{attribute 'linkalways'} 
{attribute 'no_explicit_call' := 'This FB is a CLASS and must be accessed using methods or properties'}
{attribute 'enable_dynamic_creation'}
FUNCTION_BLOCK Node_F_VN_ContourMoments EXTENDS VisionNode
VAR
    ipContour : _ITcVnContainer;
    stMoments : _TcVnMoments;
    hrPrev : _HRESULT(S_OK);
	hresult : _HRESULT(S_OK);
END_VAR

METHOD PUBLIC  Clone : I_Node
VAR
	pNode : POINTER TO Node_F_VN_ContourMoments;
END_VAR
pNode := __NEW(Node_F_VN_ContourMoments);
Clone := pNode^;
END_METHOD

METHOD FB_init : BOOL
VAR_INPUT
	bInitRetains : BOOL; // if TRUE, the retain variables are initialized (warm start / cold start)
	bInCopyCode : BOOL;  // if TRUE, the instance afterwards gets moved into the copy code (online change)
END_VAR
AddInput('ipContour', ipContour);
AddInput('hrPrev', hrPrev);
AddOutput('stMoments', stMoments);
AddOutput('hresult',hresult);
END_METHOD

METHOD PROTECTED OnExecute
hresult.Value := F_VN_ContourMoments(
	ipContour := ipContour.Value,
    stMoments := stMoments.Value,
	hrPrev:= hrPrev.Value);
END_METHOD

METHOD PUBLIC PreExecutionCheck
VAR_INPUT
	Check : I_PreExecutionChecks;
END_VAR
Check.IsTrue(ipContour.IsValid, 'ipContour must be a valid container');
Check.IsTrue((ipContour.IsType(TC_GLOBAL_CONST_LIST.ContainerType_Vector_TcVnPoint2_DINT) OR
              ipContour.IsType(TC_GLOBAL_CONST_LIST.ContainerType_Vector_TcVnPoint2_REAL)),
              'ipContour contains incorrect type');
END_METHOD

END_FUNCTION_BLOCK

(* stored: Version 1.1.0.1, ProductVersion 3.1.4026.13
   POU Node_F_VN_ContourMoments: Id {f1f8bd5b-fb7d-09f7-3cd6-ff0fb48e97c2}, SpecialFunc None
   Folder Constructor: Id {1bb0c863-8b3a-0ade-09be-99531624ab88}
   Method Clone: Id {44b8e371-313f-0c62-0852-1be687f9b1b8}
   Method FB_init: Id {a5f4f229-2a67-036c-16f2-5f92c8fbdc9f}
   Method OnExecute: Id {c4c36102-abd8-06bc-07cb-461d12efa5b6}
   Method PreExecutionCheck: Id {41b2994d-04db-09ab-2716-11f969b83f40} *)
